{attribute 'GeneratedUsingTerminal: EK1100-0000-0018'}
{attribute addProperty BoxType "EK1100-0000-0018"}
{attribute addProperty Id "Beckhoff_ELM3xxx_0030EK1122Beckhoff_ELM3xxx_0030EK1122_7B8BEA862A_0001_ELM3002_0030_0017ELM3002_73CCAB7A50A_0002_ELM3002_0030_0018ELM3002_73CCAB7A50A_0003_ELM3004_0030_0018ELM3004_7474644C72A_0004_ELM3004_0030_0019ELM3004_7474644C72A_0005_ELM3502_0030_0019ELM3502_73CCAB7A50A_0006_ELM3504_0030_0019ELM3504_7474644C72"}
{attribute addProperty CRC "1970588949"}
{attribute addProperty Size "368"}
TYPE Beckhoff_ELM3xxx_0030_7574CD15 EXTENDS EK1100_AB5A9467 :
STRUCT
	{attribute addProperty Name "Beckhoff_ELM3xxx_0030EK1122"}
	Beckhoff_ELM3xxx_0030EK1122 : Beckhoff_ELM3xxx_0030EK1122_7B8BEA86;
	{attribute addProperty Name "A_0001_ELM3002_0030_0017"}
	A_0001_ELM3002_0030_0017 : ELM3002_73CCAB7A;
	{attribute addProperty Name "A_0002_ELM3002_0030_0018"}
	A_0002_ELM3002_0030_0018 : ELM3002_73CCAB7A;
	{attribute addProperty Name "A_0003_ELM3004_0030_0018"}
	A_0003_ELM3004_0030_0018 : ELM3004_7474644C;
	{attribute addProperty Name "A_0004_ELM3004_0030_0019"}
	A_0004_ELM3004_0030_0019 : ELM3004_7474644C;
	{attribute addProperty Name "A_0005_ELM3502_0030_0019"}
	A_0005_ELM3502_0030_0019 : ELM3502_73CCAB7A;
	{attribute addProperty Name "A_0006_ELM3504_0030_0019"}
	A_0006_ELM3504_0030_0019 : ELM3504_7474644C;
END_STRUCT
END_TYPE

(* stored: Version 1.2.0.0, ProductVersion 3.1.4024.9
   DUT Beckhoff_ELM3xxx_0030_7574CD15: Id {4482e398-8ea9-469a-9926-f4180637d51b} *)
